TYPE ST_Fenster_Stellwert :
STRUCT
	Freigabe		: BOOL;
	Stellung		: BOOL;

	Fenster_AUF		: BOOL;
	Fenster_ZU		: BOOL;




END_STRUCT
END_TYPE

(* stored: Version 1.1.0.1, ProductVersion 3.1.4024.9
   DUT ST_Fenster_Stellwert: Id {c62d297c-76a6-4fa9-9cec-9c7f45b3926a} *)
